KUKA KRL data list: motion_and_splines.dat

&ACCESS RVP
&REL 1
DEFDAT motion_and_splines
  DECL E6POS xLinPoint1 = {X 1200.0, Y -300.0, Z 800.0, A 0.0, B 90.0, C 0.0, S 2, T 35}
  DECL E6POS xLinPoint2 = {X 1200.0, Y 300.0, Z 800.0, A 0.0, B 90.0, C 0.0, S 2, T 35}
  DECL E6POS xCircAux = {X 1250.0, Y 0.0, Z 850.0, A 0.0, B 90.0, C 0.0, S 2, T 35}
  DECL E6POS xCircEnd = {X 1300.0, Y -300.0, Z 800.0, A 0.0, B 90.0, C 0.0, S 2, T 35}

  ; Motion inline form companion variables
  DECL E6AXIS XHOME = {A1 0.0, A2 -90.0, A3 90.0, A4 0.0, A5 45.0, A6 0.0, E1 0.0}
  DECL FDAT fHOME = {TOOL_NO 1, BASE_NO 0, IPO_FRAME #BASE}
  DECL PDAT PPDAT1 = {VEL 100.0, ACC 100.0, APO_DIST 100.0}
  DECL E6POS XP1 = {X 1100.0, Y 0.0, Z 750.0, A 0.0, B 90.0, C 0.0, S 2, T 35}
  DECL FDAT fP1 = {TOOL_NO 1, BASE_NO 0, IPO_FRAME #BASE}
  DECL LDAT LCPDAT1 = {VEL 2.0, ACC 100.0, APO_DIST 100.0, APO_FAC 50.0}
  DECL E6POS XP_AUX = {X 1150.0, Y 50.0, Z 770.0, A 0.0, B 90.0, C 0.0, S 2, T 35}
  DECL E6POS XP2 = {X 1200.0, Y 100.0, Z 800.0, A 0.0, B 90.0, C 0.0, S 2, T 35}
  DECL FDAT fP2 = {TOOL_NO 1, BASE_NO 0, IPO_FRAME #BASE}
ENDDAT
